# EPICS substitutions: viocs/si_bpms/si_bpmsApp/Db/bpm.substitutions
file "db/bpm.db" {
    pattern { sector, pos }

        { "01", "M1" }
        { "01", "M2" }
        { "01", "C1-A" }
        { "01", "C1-B" }
        { "01", "C2-A" }
        { "01", "C2-B" }
        { "01", "C3-A" }
        { "01", "C3-B" }
        { "01", "C4" }

        { "02", "M1" }
        { "02", "M2" }
        { "02", "C1-A" }
        { "02", "C1-B" }
        { "02", "C2-A" }
        { "02", "C2-B" }
        { "02", "C3-A" }
        { "02", "C3-B" }
        { "02", "C4" }

        { "03", "M1" }
        { "03", "M2" }
        { "03", "C1-A" }
        { "03", "C1-B" }
        { "03", "C2-A" }
        { "03", "C2-B" }
        { "03", "C3-A" }
        { "03", "C3-B" }
        { "03", "C4" }

        { "04", "M1" }
        { "04", "M2" }
        { "04", "C1-A" }
        { "04", "C1-B" }
        { "04", "C2-A" }
        { "04", "C2-B" }
        { "04", "C3-A" }
        { "04", "C3-B" }
        { "04", "C4" }

        { "05", "M1" }
        { "05", "M2" }
        { "05", "C1-A" }
        { "05", "C1-B" }
        { "05", "C2-A" }
        { "05", "C2-B" }
        { "05", "C3-A" }
        { "05", "C3-B" }
        { "05", "C4" }

        { "06", "M1" }
        { "06", "M2" }
        { "06", "C1-A" }
        { "06", "C1-B" }
        { "06", "C2-A" }
        { "06", "C2-B" }
        { "06", "C3-A" }
        { "06", "C3-B" }
        { "06", "C4" }

        { "07", "M1" }
        { "07", "M2" }
        { "07", "C1-A" }
        { "07", "C1-B" }
        { "07", "C2-A" }
        { "07", "C2-B" }
        { "07", "C3-A" }
        { "07", "C3-B" }
        { "07", "C4" }

        { "08", "M1" }
        { "08", "M2" }
        { "08", "C1-A" }
        { "08", "C1-B" }
        { "08", "C2-A" }
        { "08", "C2-B" }
        { "08", "C3-A" }
        { "08", "C3-B" }
        { "08", "C4" }

        { "09", "M1" }
        { "09", "M2" }
        { "09", "C1-A" }
        { "09", "C1-B" }
        { "09", "C2-A" }
        { "09", "C2-B" }
        { "09", "C3-A" }
        { "09", "C3-B" }
        { "09", "C4" }

        { "10", "M1" }
        { "10", "M2" }
        { "10", "C1-A" }
        { "10", "C1-B" }
        { "10", "C2-A" }
        { "10", "C2-B" }
        { "10", "C3-A" }
        { "10", "C3-B" }
        { "10", "C4" }

        { "11", "M1" }
        { "11", "M2" }
        { "11", "C1-A" }
        { "11", "C1-B" }
        { "11", "C2-A" }
        { "11", "C2-B" }
        { "11", "C3-A" }
        { "11", "C3-B" }
        { "11", "C4" }

        { "12", "M1" }
        { "12", "M2" }
        { "12", "C1-A" }
        { "12", "C1-B" }
        { "12", "C2-A" }
        { "12", "C2-B" }
        { "12", "C3-A" }
        { "12", "C3-B" }
        { "12", "C4" }

        { "13", "M1" }
        { "13", "M2" }
        { "13", "C1-A" }
        { "13", "C1-B" }
        { "13", "C2-A" }
        { "13", "C2-B" }
        { "13", "C3-A" }
        { "13", "C3-B" }
        { "13", "C4" }

        { "14", "M1" }
        { "14", "M2" }
        { "14", "C1-A" }
        { "14", "C1-B" }
        { "14", "C2-A" }
        { "14", "C2-B" }
        { "14", "C3-A" }
        { "14", "C3-B" }
        { "14", "C4" }

        { "15", "M1" }
        { "15", "M2" }
        { "15", "C1-A" }
        { "15", "C1-B" }
        { "15", "C2-A" }
        { "15", "C2-B" }
        { "15", "C3-A" }
        { "15", "C3-B" }
        { "15", "C4" }

        { "16", "M1" }
        { "16", "M2" }
        { "16", "C1-A" }
        { "16", "C1-B" }
        { "16", "C2-A" }
        { "16", "C2-B" }
        { "16", "C3-A" }
        { "16", "C3-B" }
        { "16", "C4" }

        { "17", "M1" }
        { "17", "M2" }
        { "17", "C1-A" }
        { "17", "C1-B" }
        { "17", "C2-A" }
        { "17", "C2-B" }
        { "17", "C3-A" }
        { "17", "C3-B" }
        { "17", "C4" }

        { "18", "M1" }
        { "18", "M2" }
        { "18", "C1-A" }
        { "18", "C1-B" }
        { "18", "C2-A" }
        { "18", "C2-B" }
        { "18", "C3-A" }
        { "18", "C3-B" }
        { "18", "C4" }

        { "19", "M1" }
        { "19", "M2" }
        { "19", "C1-A" }
        { "19", "C1-B" }
        { "19", "C2-A" }
        { "19", "C2-B" }
        { "19", "C3-A" }
        { "19", "C3-B" }
        { "19", "C4" }

        { "20", "M1" }
        { "20", "M2" }
        { "20", "C1-A" }
        { "20", "C1-B" }
        { "20", "C2-A" }
        { "20", "C2-B" }
        { "20", "C3-A" }
        { "20", "C3-B" }
        { "20", "C4" }

}
